(* IEC 61131-3 sources: TIA2AX/tests/test_projects/expected/HW_2000482_V18/6A1_AS17, 6 files *)

(* ---- HwInputs.st ---- *)
TYPE
	HwInputs : STRUCT
		_6A2_AS17_6A3 AT %B0 : WORD;
		_6A2_AS17_6A4 AT %B2 : WORD;
		_6A2_AS17_6A13 AT %B113 : ARRAY[0..31] OF BYTE;
		_6A2_AS17_6A20 AT %B30 : ARRAY[0..7] OF BYTE;
		HousingReader_AS17_Handshake_and_General_Error_Status_Bits_1 AT %B51 : BYTE;
		HousingReader_AS17_BUSY_Status_Bits_1 AT %B52 : BYTE;
		HousingReader_AS17_Completion_Status_Bits_1 AT %B53 : BYTE;
		HousingReader_AS17_Error_Status_Bits_1 AT %B54 : BYTE;
		HousingReader_AS17_Terminal_Status_Bits_1 AT %B55 : BYTE;
		HousingReader_AS17_Unstable_Read_Status_Bits_1 AT %B56 : BYTE;
		HousingReader_AS17_Matching_Level_and_Total_Evaluation_Grade_Status_1 AT %B57 : ARRAY[0..7] OF BYTE;
		HousingReader_AS17_Operation_Result_Status_1 AT %B87 : ARRAY[0..19] OF BYTE;
		HousingReader_AS17_Read_Data_128Byte_1 AT %B229 : ARRAY[0..135] OF BYTE;
		SEW_AS_1_Drive_1x3PD_1 AT %B107 : ARRAY[0..5] OF BYTE;
		Glue_DI_16_bytes_1 AT %B65 : ARRAY[0..15] OF BYTE;
		wp12_wp12 AT %B4 : BYTE;
	END_STRUCT;
END_TYPE

(* ---- HwOutputs.st ---- *)
TYPE
	HwOutputs : STRUCT
		_6A2_AS17_6A5 AT %B0 : WORD;
		_6A2_AS17_6A6 AT %B2 : WORD;
		_6A2_AS17_6A13 AT %B87 : ARRAY[0..31] OF BYTE;
		HousingReader_AS17_Latch_and_Error_Clear_Control_Bits_1 AT %B6 : BYTE;
		HousingReader_AS17_Operation_instruction_Control_Bits_1 AT %B7 : BYTE;
		HousingReader_AS17_Completion_Clear_Control_Bits_1 AT %B12 : BYTE;
		HousingReader_AS17_Parameter_Bank_Number_1 AT %B51 : WORD;
		HousingReader_AS17_User_Data_128Byte_1 AT %B193 : ARRAY[0..129] OF BYTE;
		CPX_PneuOst_AS17_MPA1S_VMPA1_FB_EMS_8_8DO_1 AT %B13 : BYTE;
		CPX_PneuOst_AS17_MPA1S_VMPA1_FB_EMS_8_8DO_2 AT %B183 : BYTE;
		CPX_PneuOst_AS17_MPA1S_VMPA1_FB_EMS_8_8DO_3 AT %B184 : BYTE;
		CPX_PneuOst_AS17_MPA1S_VMPA1_FB_EMS_8_8DO_4 AT %B185 : BYTE;
		CPX_PneuOst_AS17_MPA1G_VMPA1_FB_EMG_8_8DO_1 AT %B4 : BYTE;
		SEW_AS_1_Drive_1x3PD_1 AT %B69 : ARRAY[0..5] OF BYTE;
		Glue_DO_16_bytes_1 AT %B30 : ARRAY[0..15] OF BYTE;
	END_STRUCT;
END_TYPE

(* ---- PlcInputs.st ---- *)
TYPE
	PlcInputs : STRUCT
		_6A2_AS17_6A3 : WORD;
		_6A2_AS17_6A4 : WORD;
		_6A2_AS17_6A13 : ARRAY[0..31] OF BYTE;
		_6A2_AS17_6A20 : ARRAY[0..7] OF BYTE;
		HousingReader_AS17_Handshake_and_General_Error_Status_Bits_1 : BYTE;
		HousingReader_AS17_BUSY_Status_Bits_1 : BYTE;
		HousingReader_AS17_Completion_Status_Bits_1 : BYTE;
		HousingReader_AS17_Error_Status_Bits_1 : BYTE;
		HousingReader_AS17_Terminal_Status_Bits_1 : BYTE;
		HousingReader_AS17_Unstable_Read_Status_Bits_1 : BYTE;
		HousingReader_AS17_Matching_Level_and_Total_Evaluation_Grade_Status_1 : ARRAY[0..7] OF BYTE;
		HousingReader_AS17_Operation_Result_Status_1 : ARRAY[0..19] OF BYTE;
		HousingReader_AS17_Read_Data_128Byte_1 : ARRAY[0..135] OF BYTE;
		SEW_AS_1_Drive_1x3PD_1 : ARRAY[0..5] OF BYTE;
		Glue_DI_16_bytes_1 : ARRAY[0..15] OF BYTE;
		wp12_wp12 : BYTE;
	END_STRUCT;
END_TYPE

(* ---- PlcOutputs.st ---- *)
TYPE
	PlcOutputs : STRUCT
		_6A2_AS17_6A5 : WORD;
		_6A2_AS17_6A6 : WORD;
		_6A2_AS17_6A13 : ARRAY[0..31] OF BYTE;
		HousingReader_AS17_Latch_and_Error_Clear_Control_Bits_1 : BYTE;
		HousingReader_AS17_Operation_instruction_Control_Bits_1 : BYTE;
		HousingReader_AS17_Completion_Clear_Control_Bits_1 : BYTE;
		HousingReader_AS17_Parameter_Bank_Number_1 : WORD;
		HousingReader_AS17_User_Data_128Byte_1 : ARRAY[0..129] OF BYTE;
		CPX_PneuOst_AS17_MPA1S_VMPA1_FB_EMS_8_8DO_1 : BYTE;
		CPX_PneuOst_AS17_MPA1S_VMPA1_FB_EMS_8_8DO_2 : BYTE;
		CPX_PneuOst_AS17_MPA1S_VMPA1_FB_EMS_8_8DO_3 : BYTE;
		CPX_PneuOst_AS17_MPA1S_VMPA1_FB_EMS_8_8DO_4 : BYTE;
		CPX_PneuOst_AS17_MPA1G_VMPA1_FB_EMG_8_8DO_1 : BYTE;
		SEW_AS_1_Drive_1x3PD_1 : ARRAY[0..5] OF BYTE;
		Glue_DO_16_bytes_1 : ARRAY[0..15] OF BYTE;
	END_STRUCT;
END_TYPE

(* ---- CopyInputs.st ---- *)
FUNCTION CopyInputs
	VAR_EXTERNAL
		HwInputs : HwInputs;
		PlcInputs : PlcInputs;
	END_VAR
	PlcInputs._6A2_AS17_6A3 := HwInputs._6A2_AS17_6A3;
	PlcInputs._6A2_AS17_6A4 := HwInputs._6A2_AS17_6A4;
	PlcInputs._6A2_AS17_6A13[0] := HwInputs._6A2_AS17_6A13[0];
	PlcInputs._6A2_AS17_6A13[1] := HwInputs._6A2_AS17_6A13[1];
	PlcInputs._6A2_AS17_6A13[2] := HwInputs._6A2_AS17_6A13[2];
	PlcInputs._6A2_AS17_6A13[3] := HwInputs._6A2_AS17_6A13[3];
	PlcInputs._6A2_AS17_6A13[4] := HwInputs._6A2_AS17_6A13[4];
	PlcInputs._6A2_AS17_6A13[5] := HwInputs._6A2_AS17_6A13[5];
	PlcInputs._6A2_AS17_6A13[6] := HwInputs._6A2_AS17_6A13[6];
	PlcInputs._6A2_AS17_6A13[7] := HwInputs._6A2_AS17_6A13[7];
	PlcInputs._6A2_AS17_6A13[8] := HwInputs._6A2_AS17_6A13[8];
	PlcInputs._6A2_AS17_6A13[9] := HwInputs._6A2_AS17_6A13[9];
	PlcInputs._6A2_AS17_6A13[10] := HwInputs._6A2_AS17_6A13[10];
	PlcInputs._6A2_AS17_6A13[11] := HwInputs._6A2_AS17_6A13[11];
	PlcInputs._6A2_AS17_6A13[12] := HwInputs._6A2_AS17_6A13[12];
	PlcInputs._6A2_AS17_6A13[13] := HwInputs._6A2_AS17_6A13[13];
	PlcInputs._6A2_AS17_6A13[14] := HwInputs._6A2_AS17_6A13[14];
	PlcInputs._6A2_AS17_6A13[15] := HwInputs._6A2_AS17_6A13[15];
	PlcInputs._6A2_AS17_6A13[16] := HwInputs._6A2_AS17_6A13[16];
	PlcInputs._6A2_AS17_6A13[17] := HwInputs._6A2_AS17_6A13[17];
	PlcInputs._6A2_AS17_6A13[18] := HwInputs._6A2_AS17_6A13[18];
	PlcInputs._6A2_AS17_6A13[19] := HwInputs._6A2_AS17_6A13[19];
	PlcInputs._6A2_AS17_6A13[20] := HwInputs._6A2_AS17_6A13[20];
	PlcInputs._6A2_AS17_6A13[21] := HwInputs._6A2_AS17_6A13[21];
	PlcInputs._6A2_AS17_6A13[22] := HwInputs._6A2_AS17_6A13[22];
	PlcInputs._6A2_AS17_6A13[23] := HwInputs._6A2_AS17_6A13[23];
	PlcInputs._6A2_AS17_6A13[24] := HwInputs._6A2_AS17_6A13[24];
	PlcInputs._6A2_AS17_6A13[25] := HwInputs._6A2_AS17_6A13[25];
	PlcInputs._6A2_AS17_6A13[26] := HwInputs._6A2_AS17_6A13[26];
	PlcInputs._6A2_AS17_6A13[27] := HwInputs._6A2_AS17_6A13[27];
	PlcInputs._6A2_AS17_6A13[28] := HwInputs._6A2_AS17_6A13[28];
	PlcInputs._6A2_AS17_6A13[29] := HwInputs._6A2_AS17_6A13[29];
	PlcInputs._6A2_AS17_6A13[30] := HwInputs._6A2_AS17_6A13[30];
	PlcInputs._6A2_AS17_6A13[31] := HwInputs._6A2_AS17_6A13[31];
	PlcInputs._6A2_AS17_6A20[0] := HwInputs._6A2_AS17_6A20[0];
	PlcInputs._6A2_AS17_6A20[1] := HwInputs._6A2_AS17_6A20[1];
	PlcInputs._6A2_AS17_6A20[2] := HwInputs._6A2_AS17_6A20[2];
	PlcInputs._6A2_AS17_6A20[3] := HwInputs._6A2_AS17_6A20[3];
	PlcInputs._6A2_AS17_6A20[4] := HwInputs._6A2_AS17_6A20[4];
	PlcInputs._6A2_AS17_6A20[5] := HwInputs._6A2_AS17_6A20[5];
	PlcInputs._6A2_AS17_6A20[6] := HwInputs._6A2_AS17_6A20[6];
	PlcInputs._6A2_AS17_6A20[7] := HwInputs._6A2_AS17_6A20[7];
	PlcInputs.HousingReader_AS17_Handshake_and_General_Error_Status_Bits_1 := HwInputs.HousingReader_AS17_Handshake_and_General_Error_Status_Bits_1;
	PlcInputs.HousingReader_AS17_BUSY_Status_Bits_1 := HwInputs.HousingReader_AS17_BUSY_Status_Bits_1;
	PlcInputs.HousingReader_AS17_Completion_Status_Bits_1 := HwInputs.HousingReader_AS17_Completion_Status_Bits_1;
	PlcInputs.HousingReader_AS17_Error_Status_Bits_1 := HwInputs.HousingReader_AS17_Error_Status_Bits_1;
	PlcInputs.HousingReader_AS17_Terminal_Status_Bits_1 := HwInputs.HousingReader_AS17_Terminal_Status_Bits_1;
	PlcInputs.HousingReader_AS17_Unstable_Read_Status_Bits_1 := HwInputs.HousingReader_AS17_Unstable_Read_Status_Bits_1;
	PlcInputs.HousingReader_AS17_Matching_Level_and_Total_Evaluation_Grade_Status_1[0] := HwInputs.HousingReader_AS17_Matching_Level_and_Total_Evaluation_Grade_Status_1[0];
	PlcInputs.HousingReader_AS17_Matching_Level_and_Total_Evaluation_Grade_Status_1[1] := HwInputs.HousingReader_AS17_Matching_Level_and_Total_Evaluation_Grade_Status_1[1];
	PlcInputs.HousingReader_AS17_Matching_Level_and_Total_Evaluation_Grade_Status_1[2] := HwInputs.HousingReader_AS17_Matching_Level_and_Total_Evaluation_Grade_Status_1[2];
	PlcInputs.HousingReader_AS17_Matching_Level_and_Total_Evaluation_Grade_Status_1[3] := HwInputs.HousingReader_AS17_Matching_Level_and_Total_Evaluation_Grade_Status_1[3];
	PlcInputs.HousingReader_AS17_Matching_Level_and_Total_Evaluation_Grade_Status_1[4] := HwInputs.HousingReader_AS17_Matching_Level_and_Total_Evaluation_Grade_Status_1[4];
	PlcInputs.HousingReader_AS17_Matching_Level_and_Total_Evaluation_Grade_Status_1[5] := HwInputs.HousingReader_AS17_Matching_Level_and_Total_Evaluation_Grade_Status_1[5];
	PlcInputs.HousingReader_AS17_Matching_Level_and_Total_Evaluation_Grade_Status_1[6] := HwInputs.HousingReader_AS17_Matching_Level_and_Total_Evaluation_Grade_Status_1[6];
	PlcInputs.HousingReader_AS17_Matching_Level_and_Total_Evaluation_Grade_Status_1[7] := HwInputs.HousingReader_AS17_Matching_Level_and_Total_Evaluation_Grade_Status_1[7];
	PlcInputs.HousingReader_AS17_Operation_Result_Status_1[0] := HwInputs.HousingReader_AS17_Operation_Result_Status_1[0];
	PlcInputs.HousingReader_AS17_Operation_Result_Status_1[1] := HwInputs.HousingReader_AS17_Operation_Result_Status_1[1];
	PlcInputs.HousingReader_AS17_Operation_Result_Status_1[2] := HwInputs.HousingReader_AS17_Operation_Result_Status_1[2];
	PlcInputs.HousingReader_AS17_Operation_Result_Status_1[3] := HwInputs.HousingReader_AS17_Operation_Result_Status_1[3];
	PlcInputs.HousingReader_AS17_Operation_Result_Status_1[4] := HwInputs.HousingReader_AS17_Operation_Result_Status_1[4];
	PlcInputs.HousingReader_AS17_Operation_Result_Status_1[5] := HwInputs.HousingReader_AS17_Operation_Result_Status_1[5];
	PlcInputs.HousingReader_AS17_Operation_Result_Status_1[6] := HwInputs.HousingReader_AS17_Operation_Result_Status_1[6];
	PlcInputs.HousingReader_AS17_Operation_Result_Status_1[7] := HwInputs.HousingReader_AS17_Operation_Result_Status_1[7];
	PlcInputs.HousingReader_AS17_Operation_Result_Status_1[8] := HwInputs.HousingReader_AS17_Operation_Result_Status_1[8];
	PlcInputs.HousingReader_AS17_Operation_Result_Status_1[9] := HwInputs.HousingReader_AS17_Operation_Result_Status_1[9];
	PlcInputs.HousingReader_AS17_Operation_Result_Status_1[10] := HwInputs.HousingReader_AS17_Operation_Result_Status_1[10];
	PlcInputs.HousingReader_AS17_Operation_Result_Status_1[11] := HwInputs.HousingReader_AS17_Operation_Result_Status_1[11];
	PlcInputs.HousingReader_AS17_Operation_Result_Status_1[12] := HwInputs.HousingReader_AS17_Operation_Result_Status_1[12];
	PlcInputs.HousingReader_AS17_Operation_Result_Status_1[13] := HwInputs.HousingReader_AS17_Operation_Result_Status_1[13];
	PlcInputs.HousingReader_AS17_Operation_Result_Status_1[14] := HwInputs.HousingReader_AS17_Operation_Result_Status_1[14];
	PlcInputs.HousingReader_AS17_Operation_Result_Status_1[15] := HwInputs.HousingReader_AS17_Operation_Result_Status_1[15];
	PlcInputs.HousingReader_AS17_Operation_Result_Status_1[16] := HwInputs.HousingReader_AS17_Operation_Result_Status_1[16];
	PlcInputs.HousingReader_AS17_Operation_Result_Status_1[17] := HwInputs.HousingReader_AS17_Operation_Result_Status_1[17];
	PlcInputs.HousingReader_AS17_Operation_Result_Status_1[18] := HwInputs.HousingReader_AS17_Operation_Result_Status_1[18];
	PlcInputs.HousingReader_AS17_Operation_Result_Status_1[19] := HwInputs.HousingReader_AS17_Operation_Result_Status_1[19];
	PlcInputs.HousingReader_AS17_Read_Data_128Byte_1[0] := HwInputs.HousingReader_AS17_Read_Data_128Byte_1[0];
	PlcInputs.HousingReader_AS17_Read_Data_128Byte_1[1] := HwInputs.HousingReader_AS17_Read_Data_128Byte_1[1];
	PlcInputs.HousingReader_AS17_Read_Data_128Byte_1[2] := HwInputs.HousingReader_AS17_Read_Data_128Byte_1[2];
	PlcInputs.HousingReader_AS17_Read_Data_128Byte_1[3] := HwInputs.HousingReader_AS17_Read_Data_128Byte_1[3];
	PlcInputs.HousingReader_AS17_Read_Data_128Byte_1[4] := HwInputs.HousingReader_AS17_Read_Data_128Byte_1[4];
	PlcInputs.HousingReader_AS17_Read_Data_128Byte_1[5] := HwInputs.HousingReader_AS17_Read_Data_128Byte_1[5];
	PlcInputs.HousingReader_AS17_Read_Data_128Byte_1[6] := HwInputs.HousingReader_AS17_Read_Data_128Byte_1[6];
	PlcInputs.HousingReader_AS17_Read_Data_128Byte_1[7] := HwInputs.HousingReader_AS17_Read_Data_128Byte_1[7];
	PlcInputs.HousingReader_AS17_Read_Data_128Byte_1[8] := HwInputs.HousingReader_AS17_Read_Data_128Byte_1[8];
	PlcInputs.HousingReader_AS17_Read_Data_128Byte_1[9] := HwInputs.HousingReader_AS17_Read_Data_128Byte_1[9];
	PlcInputs.HousingReader_AS17_Read_Data_128Byte_1[10] := HwInputs.HousingReader_AS17_Read_Data_128Byte_1[10];
	PlcInputs.HousingReader_AS17_Read_Data_128Byte_1[11] := HwInputs.HousingReader_AS17_Read_Data_128Byte_1[11];
	PlcInputs.HousingReader_AS17_Read_Data_128Byte_1[12] := HwInputs.HousingReader_AS17_Read_Data_128Byte_1[12];
	PlcInputs.HousingReader_AS17_Read_Data_128Byte_1[13] := HwInputs.HousingReader_AS17_Read_Data_128Byte_1[13];
	PlcInputs.HousingReader_AS17_Read_Data_128Byte_1[14] := HwInputs.HousingReader_AS17_Read_Data_128Byte_1[14];
	PlcInputs.HousingReader_AS17_Read_Data_128Byte_1[15] := HwInputs.HousingReader_AS17_Read_Data_128Byte_1[15];
	PlcInputs.HousingReader_AS17_Read_Data_128Byte_1[16] := HwInputs.HousingReader_AS17_Read_Data_128Byte_1[16];
	PlcInputs.HousingReader_AS17_Read_Data_128Byte_1[17] := HwInputs.HousingReader_AS17_Read_Data_128Byte_1[17];
	PlcInputs.HousingReader_AS17_Read_Data_128Byte_1[18] := HwInputs.HousingReader_AS17_Read_Data_128Byte_1[18];
	PlcInputs.HousingReader_AS17_Read_Data_128Byte_1[19] := HwInputs.HousingReader_AS17_Read_Data_128Byte_1[19];
	PlcInputs.HousingReader_AS17_Read_Data_128Byte_1[20] := HwInputs.HousingReader_AS17_Read_Data_128Byte_1[20];
	PlcInputs.HousingReader_AS17_Read_Data_128Byte_1[21] := HwInputs.HousingReader_AS17_Read_Data_128Byte_1[21];
	PlcInputs.HousingReader_AS17_Read_Data_128Byte_1[22] := HwInputs.HousingReader_AS17_Read_Data_128Byte_1[22];
	PlcInputs.HousingReader_AS17_Read_Data_128Byte_1[23] := HwInputs.HousingReader_AS17_Read_Data_128Byte_1[23];
	PlcInputs.HousingReader_AS17_Read_Data_128Byte_1[24] := HwInputs.HousingReader_AS17_Read_Data_128Byte_1[24];
	PlcInputs.HousingReader_AS17_Read_Data_128Byte_1[25] := HwInputs.HousingReader_AS17_Read_Data_128Byte_1[25];
	PlcInputs.HousingReader_AS17_Read_Data_128Byte_1[26] := HwInputs.HousingReader_AS17_Read_Data_128Byte_1[26];
	PlcInputs.HousingReader_AS17_Read_Data_128Byte_1[27] := HwInputs.HousingReader_AS17_Read_Data_128Byte_1[27];
	PlcInputs.HousingReader_AS17_Read_Data_128Byte_1[28] := HwInputs.HousingReader_AS17_Read_Data_128Byte_1[28];
	PlcInputs.HousingReader_AS17_Read_Data_128Byte_1[29] := HwInputs.HousingReader_AS17_Read_Data_128Byte_1[29];
	PlcInputs.HousingReader_AS17_Read_Data_128Byte_1[30] := HwInputs.HousingReader_AS17_Read_Data_128Byte_1[30];
	PlcInputs.HousingReader_AS17_Read_Data_128Byte_1[31] := HwInputs.HousingReader_AS17_Read_Data_128Byte_1[31];
	PlcInputs.HousingReader_AS17_Read_Data_128Byte_1[32] := HwInputs.HousingReader_AS17_Read_Data_128Byte_1[32];
	PlcInputs.HousingReader_AS17_Read_Data_128Byte_1[33] := HwInputs.HousingReader_AS17_Read_Data_128Byte_1[33];
	PlcInputs.HousingReader_AS17_Read_Data_128Byte_1[34] := HwInputs.HousingReader_AS17_Read_Data_128Byte_1[34];
	PlcInputs.HousingReader_AS17_Read_Data_128Byte_1[35] := HwInputs.HousingReader_AS17_Read_Data_128Byte_1[35];
	PlcInputs.HousingReader_AS17_Read_Data_128Byte_1[36] := HwInputs.HousingReader_AS17_Read_Data_128Byte_1[36];
	PlcInputs.HousingReader_AS17_Read_Data_128Byte_1[37] := HwInputs.HousingReader_AS17_Read_Data_128Byte_1[37];
	PlcInputs.HousingReader_AS17_Read_Data_128Byte_1[38] := HwInputs.HousingReader_AS17_Read_Data_128Byte_1[38];
	PlcInputs.HousingReader_AS17_Read_Data_128Byte_1[39] := HwInputs.HousingReader_AS17_Read_Data_128Byte_1[39];
	PlcInputs.HousingReader_AS17_Read_Data_128Byte_1[40] := HwInputs.HousingReader_AS17_Read_Data_128Byte_1[40];
	PlcInputs.HousingReader_AS17_Read_Data_128Byte_1[41] := HwInputs.HousingReader_AS17_Read_Data_128Byte_1[41];
	PlcInputs.HousingReader_AS17_Read_Data_128Byte_1[42] := HwInputs.HousingReader_AS17_Read_Data_128Byte_1[42];
	PlcInputs.HousingReader_AS17_Read_Data_128Byte_1[43] := HwInputs.HousingReader_AS17_Read_Data_128Byte_1[43];
	PlcInputs.HousingReader_AS17_Read_Data_128Byte_1[44] := HwInputs.HousingReader_AS17_Read_Data_128Byte_1[44];
	PlcInputs.HousingReader_AS17_Read_Data_128Byte_1[45] := HwInputs.HousingReader_AS17_Read_Data_128Byte_1[45];
	PlcInputs.HousingReader_AS17_Read_Data_128Byte_1[46] := HwInputs.HousingReader_AS17_Read_Data_128Byte_1[46];
	PlcInputs.HousingReader_AS17_Read_Data_128Byte_1[47] := HwInputs.HousingReader_AS17_Read_Data_128Byte_1[47];
	PlcInputs.HousingReader_AS17_Read_Data_128Byte_1[48] := HwInputs.HousingReader_AS17_Read_Data_128Byte_1[48];
	PlcInputs.HousingReader_AS17_Read_Data_128Byte_1[49] := HwInputs.HousingReader_AS17_Read_Data_128Byte_1[49];
	PlcInputs.HousingReader_AS17_Read_Data_128Byte_1[50] := HwInputs.HousingReader_AS17_Read_Data_128Byte_1[50];
	PlcInputs.HousingReader_AS17_Read_Data_128Byte_1[51] := HwInputs.HousingReader_AS17_Read_Data_128Byte_1[51];
	PlcInputs.HousingReader_AS17_Read_Data_128Byte_1[52] := HwInputs.HousingReader_AS17_Read_Data_128Byte_1[52];
	PlcInputs.HousingReader_AS17_Read_Data_128Byte_1[53] := HwInputs.HousingReader_AS17_Read_Data_128Byte_1[53];
	PlcInputs.HousingReader_AS17_Read_Data_128Byte_1[54] := HwInputs.HousingReader_AS17_Read_Data_128Byte_1[54];
	PlcInputs.HousingReader_AS17_Read_Data_128Byte_1[55] := HwInputs.HousingReader_AS17_Read_Data_128Byte_1[55];
	PlcInputs.HousingReader_AS17_Read_Data_128Byte_1[56] := HwInputs.HousingReader_AS17_Read_Data_128Byte_1[56];
	PlcInputs.HousingReader_AS17_Read_Data_128Byte_1[57] := HwInputs.HousingReader_AS17_Read_Data_128Byte_1[57];
	PlcInputs.HousingReader_AS17_Read_Data_128Byte_1[58] := HwInputs.HousingReader_AS17_Read_Data_128Byte_1[58];
	PlcInputs.HousingReader_AS17_Read_Data_128Byte_1[59] := HwInputs.HousingReader_AS17_Read_Data_128Byte_1[59];
	PlcInputs.HousingReader_AS17_Read_Data_128Byte_1[60] := HwInputs.HousingReader_AS17_Read_Data_128Byte_1[60];
	PlcInputs.HousingReader_AS17_Read_Data_128Byte_1[61] := HwInputs.HousingReader_AS17_Read_Data_128Byte_1[61];
	PlcInputs.HousingReader_AS17_Read_Data_128Byte_1[62] := HwInputs.HousingReader_AS17_Read_Data_128Byte_1[62];
	PlcInputs.HousingReader_AS17_Read_Data_128Byte_1[63] := HwInputs.HousingReader_AS17_Read_Data_128Byte_1[63];
	PlcInputs.HousingReader_AS17_Read_Data_128Byte_1[64] := HwInputs.HousingReader_AS17_Read_Data_128Byte_1[64];
	PlcInputs.HousingReader_AS17_Read_Data_128Byte_1[65] := HwInputs.HousingReader_AS17_Read_Data_128Byte_1[65];
	PlcInputs.HousingReader_AS17_Read_Data_128Byte_1[66] := HwInputs.HousingReader_AS17_Read_Data_128Byte_1[66];
	PlcInputs.HousingReader_AS17_Read_Data_128Byte_1[67] := HwInputs.HousingReader_AS17_Read_Data_128Byte_1[67];
	PlcInputs.HousingReader_AS17_Read_Data_128Byte_1[68] := HwInputs.HousingReader_AS17_Read_Data_128Byte_1[68];
	PlcInputs.HousingReader_AS17_Read_Data_128Byte_1[69] := HwInputs.HousingReader_AS17_Read_Data_128Byte_1[69];
	PlcInputs.HousingReader_AS17_Read_Data_128Byte_1[70] := HwInputs.HousingReader_AS17_Read_Data_128Byte_1[70];
	PlcInputs.HousingReader_AS17_Read_Data_128Byte_1[71] := HwInputs.HousingReader_AS17_Read_Data_128Byte_1[71];
	PlcInputs.HousingReader_AS17_Read_Data_128Byte_1[72] := HwInputs.HousingReader_AS17_Read_Data_128Byte_1[72];
	PlcInputs.HousingReader_AS17_Read_Data_128Byte_1[73] := HwInputs.HousingReader_AS17_Read_Data_128Byte_1[73];
	PlcInputs.HousingReader_AS17_Read_Data_128Byte_1[74] := HwInputs.HousingReader_AS17_Read_Data_128Byte_1[74];
	PlcInputs.HousingReader_AS17_Read_Data_128Byte_1[75] := HwInputs.HousingReader_AS17_Read_Data_128Byte_1[75];
	PlcInputs.HousingReader_AS17_Read_Data_128Byte_1[76] := HwInputs.HousingReader_AS17_Read_Data_128Byte_1[76];
	PlcInputs.HousingReader_AS17_Read_Data_128Byte_1[77] := HwInputs.HousingReader_AS17_Read_Data_128Byte_1[77];
	PlcInputs.HousingReader_AS17_Read_Data_128Byte_1[78] := HwInputs.HousingReader_AS17_Read_Data_128Byte_1[78];
	PlcInputs.HousingReader_AS17_Read_Data_128Byte_1[79] := HwInputs.HousingReader_AS17_Read_Data_128Byte_1[79];
	PlcInputs.HousingReader_AS17_Read_Data_128Byte_1[80] := HwInputs.HousingReader_AS17_Read_Data_128Byte_1[80];
	PlcInputs.HousingReader_AS17_Read_Data_128Byte_1[81] := HwInputs.HousingReader_AS17_Read_Data_128Byte_1[81];
	PlcInputs.HousingReader_AS17_Read_Data_128Byte_1[82] := HwInputs.HousingReader_AS17_Read_Data_128Byte_1[82];
	PlcInputs.HousingReader_AS17_Read_Data_128Byte_1[83] := HwInputs.HousingReader_AS17_Read_Data_128Byte_1[83];
	PlcInputs.HousingReader_AS17_Read_Data_128Byte_1[84] := HwInputs.HousingReader_AS17_Read_Data_128Byte_1[84];
	PlcInputs.HousingReader_AS17_Read_Data_128Byte_1[85] := HwInputs.HousingReader_AS17_Read_Data_128Byte_1[85];
	PlcInputs.HousingReader_AS17_Read_Data_128Byte_1[86] := HwInputs.HousingReader_AS17_Read_Data_128Byte_1[86];
	PlcInputs.HousingReader_AS17_Read_Data_128Byte_1[87] := HwInputs.HousingReader_AS17_Read_Data_128Byte_1[87];
	PlcInputs.HousingReader_AS17_Read_Data_128Byte_1[88] := HwInputs.HousingReader_AS17_Read_Data_128Byte_1[88];
	PlcInputs.HousingReader_AS17_Read_Data_128Byte_1[89] := HwInputs.HousingReader_AS17_Read_Data_128Byte_1[89];
	PlcInputs.HousingReader_AS17_Read_Data_128Byte_1[90] := HwInputs.HousingReader_AS17_Read_Data_128Byte_1[90];
	PlcInputs.HousingReader_AS17_Read_Data_128Byte_1[91] := HwInputs.HousingReader_AS17_Read_Data_128Byte_1[91];
	PlcInputs.HousingReader_AS17_Read_Data_128Byte_1[92] := HwInputs.HousingReader_AS17_Read_Data_128Byte_1[92];
	PlcInputs.HousingReader_AS17_Read_Data_128Byte_1[93] := HwInputs.HousingReader_AS17_Read_Data_128Byte_1[93];
	PlcInputs.HousingReader_AS17_Read_Data_128Byte_1[94] := HwInputs.HousingReader_AS17_Read_Data_128Byte_1[94];
	PlcInputs.HousingReader_AS17_Read_Data_128Byte_1[95] := HwInputs.HousingReader_AS17_Read_Data_128Byte_1[95];
	PlcInputs.HousingReader_AS17_Read_Data_128Byte_1[96] := HwInputs.HousingReader_AS17_Read_Data_128Byte_1[96];
	PlcInputs.HousingReader_AS17_Read_Data_128Byte_1[97] := HwInputs.HousingReader_AS17_Read_Data_128Byte_1[97];
	PlcInputs.HousingReader_AS17_Read_Data_128Byte_1[98] := HwInputs.HousingReader_AS17_Read_Data_128Byte_1[98];
	PlcInputs.HousingReader_AS17_Read_Data_128Byte_1[99] := HwInputs.HousingReader_AS17_Read_Data_128Byte_1[99];
	PlcInputs.HousingReader_AS17_Read_Data_128Byte_1[100] := HwInputs.HousingReader_AS17_Read_Data_128Byte_1[100];
	PlcInputs.HousingReader_AS17_Read_Data_128Byte_1[101] := HwInputs.HousingReader_AS17_Read_Data_128Byte_1[101];
	PlcInputs.HousingReader_AS17_Read_Data_128Byte_1[102] := HwInputs.HousingReader_AS17_Read_Data_128Byte_1[102];
	PlcInputs.HousingReader_AS17_Read_Data_128Byte_1[103] := HwInputs.HousingReader_AS17_Read_Data_128Byte_1[103];
	PlcInputs.HousingReader_AS17_Read_Data_128Byte_1[104] := HwInputs.HousingReader_AS17_Read_Data_128Byte_1[104];
	PlcInputs.HousingReader_AS17_Read_Data_128Byte_1[105] := HwInputs.HousingReader_AS17_Read_Data_128Byte_1[105];
	PlcInputs.HousingReader_AS17_Read_Data_128Byte_1[106] := HwInputs.HousingReader_AS17_Read_Data_128Byte_1[106];
	PlcInputs.HousingReader_AS17_Read_Data_128Byte_1[107] := HwInputs.HousingReader_AS17_Read_Data_128Byte_1[107];
	PlcInputs.HousingReader_AS17_Read_Data_128Byte_1[108] := HwInputs.HousingReader_AS17_Read_Data_128Byte_1[108];
	PlcInputs.HousingReader_AS17_Read_Data_128Byte_1[109] := HwInputs.HousingReader_AS17_Read_Data_128Byte_1[109];
	PlcInputs.HousingReader_AS17_Read_Data_128Byte_1[110] := HwInputs.HousingReader_AS17_Read_Data_128Byte_1[110];
	PlcInputs.HousingReader_AS17_Read_Data_128Byte_1[111] := HwInputs.HousingReader_AS17_Read_Data_128Byte_1[111];
	PlcInputs.HousingReader_AS17_Read_Data_128Byte_1[112] := HwInputs.HousingReader_AS17_Read_Data_128Byte_1[112];
	PlcInputs.HousingReader_AS17_Read_Data_128Byte_1[113] := HwInputs.HousingReader_AS17_Read_Data_128Byte_1[113];
	PlcInputs.HousingReader_AS17_Read_Data_128Byte_1[114] := HwInputs.HousingReader_AS17_Read_Data_128Byte_1[114];
	PlcInputs.HousingReader_AS17_Read_Data_128Byte_1[115] := HwInputs.HousingReader_AS17_Read_Data_128Byte_1[115];
	PlcInputs.HousingReader_AS17_Read_Data_128Byte_1[116] := HwInputs.HousingReader_AS17_Read_Data_128Byte_1[116];
	PlcInputs.HousingReader_AS17_Read_Data_128Byte_1[117] := HwInputs.HousingReader_AS17_Read_Data_128Byte_1[117];
	PlcInputs.HousingReader_AS17_Read_Data_128Byte_1[118] := HwInputs.HousingReader_AS17_Read_Data_128Byte_1[118];
	PlcInputs.HousingReader_AS17_Read_Data_128Byte_1[119] := HwInputs.HousingReader_AS17_Read_Data_128Byte_1[119];
	PlcInputs.HousingReader_AS17_Read_Data_128Byte_1[120] := HwInputs.HousingReader_AS17_Read_Data_128Byte_1[120];
	PlcInputs.HousingReader_AS17_Read_Data_128Byte_1[121] := HwInputs.HousingReader_AS17_Read_Data_128Byte_1[121];
	PlcInputs.HousingReader_AS17_Read_Data_128Byte_1[122] := HwInputs.HousingReader_AS17_Read_Data_128Byte_1[122];
	PlcInputs.HousingReader_AS17_Read_Data_128Byte_1[123] := HwInputs.HousingReader_AS17_Read_Data_128Byte_1[123];
	PlcInputs.HousingReader_AS17_Read_Data_128Byte_1[124] := HwInputs.HousingReader_AS17_Read_Data_128Byte_1[124];
	PlcInputs.HousingReader_AS17_Read_Data_128Byte_1[125] := HwInputs.HousingReader_AS17_Read_Data_128Byte_1[125];
	PlcInputs.HousingReader_AS17_Read_Data_128Byte_1[126] := HwInputs.HousingReader_AS17_Read_Data_128Byte_1[126];
	PlcInputs.HousingReader_AS17_Read_Data_128Byte_1[127] := HwInputs.HousingReader_AS17_Read_Data_128Byte_1[127];
	PlcInputs.HousingReader_AS17_Read_Data_128Byte_1[128] := HwInputs.HousingReader_AS17_Read_Data_128Byte_1[128];
	PlcInputs.HousingReader_AS17_Read_Data_128Byte_1[129] := HwInputs.HousingReader_AS17_Read_Data_128Byte_1[129];
	PlcInputs.HousingReader_AS17_Read_Data_128Byte_1[130] := HwInputs.HousingReader_AS17_Read_Data_128Byte_1[130];
	PlcInputs.HousingReader_AS17_Read_Data_128Byte_1[131] := HwInputs.HousingReader_AS17_Read_Data_128Byte_1[131];
	PlcInputs.HousingReader_AS17_Read_Data_128Byte_1[132] := HwInputs.HousingReader_AS17_Read_Data_128Byte_1[132];
	PlcInputs.HousingReader_AS17_Read_Data_128Byte_1[133] := HwInputs.HousingReader_AS17_Read_Data_128Byte_1[133];
	PlcInputs.HousingReader_AS17_Read_Data_128Byte_1[134] := HwInputs.HousingReader_AS17_Read_Data_128Byte_1[134];
	PlcInputs.HousingReader_AS17_Read_Data_128Byte_1[135] := HwInputs.HousingReader_AS17_Read_Data_128Byte_1[135];
	PlcInputs.SEW_AS_1_Drive_1x3PD_1[0] := HwInputs.SEW_AS_1_Drive_1x3PD_1[0];
	PlcInputs.SEW_AS_1_Drive_1x3PD_1[1] := HwInputs.SEW_AS_1_Drive_1x3PD_1[1];
	PlcInputs.SEW_AS_1_Drive_1x3PD_1[2] := HwInputs.SEW_AS_1_Drive_1x3PD_1[2];
	PlcInputs.SEW_AS_1_Drive_1x3PD_1[3] := HwInputs.SEW_AS_1_Drive_1x3PD_1[3];
	PlcInputs.SEW_AS_1_Drive_1x3PD_1[4] := HwInputs.SEW_AS_1_Drive_1x3PD_1[4];
	PlcInputs.SEW_AS_1_Drive_1x3PD_1[5] := HwInputs.SEW_AS_1_Drive_1x3PD_1[5];
	PlcInputs.Glue_DI_16_bytes_1[0] := HwInputs.Glue_DI_16_bytes_1[0];
	PlcInputs.Glue_DI_16_bytes_1[1] := HwInputs.Glue_DI_16_bytes_1[1];
	PlcInputs.Glue_DI_16_bytes_1[2] := HwInputs.Glue_DI_16_bytes_1[2];
	PlcInputs.Glue_DI_16_bytes_1[3] := HwInputs.Glue_DI_16_bytes_1[3];
	PlcInputs.Glue_DI_16_bytes_1[4] := HwInputs.Glue_DI_16_bytes_1[4];
	PlcInputs.Glue_DI_16_bytes_1[5] := HwInputs.Glue_DI_16_bytes_1[5];
	PlcInputs.Glue_DI_16_bytes_1[6] := HwInputs.Glue_DI_16_bytes_1[6];
	PlcInputs.Glue_DI_16_bytes_1[7] := HwInputs.Glue_DI_16_bytes_1[7];
	PlcInputs.Glue_DI_16_bytes_1[8] := HwInputs.Glue_DI_16_bytes_1[8];
	PlcInputs.Glue_DI_16_bytes_1[9] := HwInputs.Glue_DI_16_bytes_1[9];
	PlcInputs.Glue_DI_16_bytes_1[10] := HwInputs.Glue_DI_16_bytes_1[10];
	PlcInputs.Glue_DI_16_bytes_1[11] := HwInputs.Glue_DI_16_bytes_1[11];
	PlcInputs.Glue_DI_16_bytes_1[12] := HwInputs.Glue_DI_16_bytes_1[12];
	PlcInputs.Glue_DI_16_bytes_1[13] := HwInputs.Glue_DI_16_bytes_1[13];
	PlcInputs.Glue_DI_16_bytes_1[14] := HwInputs.Glue_DI_16_bytes_1[14];
	PlcInputs.Glue_DI_16_bytes_1[15] := HwInputs.Glue_DI_16_bytes_1[15];
	PlcInputs.wp12_wp12 := HwInputs.wp12_wp12;
END_FUNCTION

(* ---- CopyOutputs.st ---- *)
FUNCTION CopyOutputs
	VAR_EXTERNAL
		HwOutputs : HwOutputs;
		PlcOutputs : PlcOutputs;
	END_VAR
	HwOutputs._6A2_AS17_6A5 := PlcOutputs._6A2_AS17_6A5;
	HwOutputs._6A2_AS17_6A6 := PlcOutputs._6A2_AS17_6A6;
	HwOutputs._6A2_AS17_6A13[0] := PlcOutputs._6A2_AS17_6A13[0];
	HwOutputs._6A2_AS17_6A13[1] := PlcOutputs._6A2_AS17_6A13[1];
	HwOutputs._6A2_AS17_6A13[2] := PlcOutputs._6A2_AS17_6A13[2];
	HwOutputs._6A2_AS17_6A13[3] := PlcOutputs._6A2_AS17_6A13[3];
	HwOutputs._6A2_AS17_6A13[4] := PlcOutputs._6A2_AS17_6A13[4];
	HwOutputs._6A2_AS17_6A13[5] := PlcOutputs._6A2_AS17_6A13[5];
	HwOutputs._6A2_AS17_6A13[6] := PlcOutputs._6A2_AS17_6A13[6];
	HwOutputs._6A2_AS17_6A13[7] := PlcOutputs._6A2_AS17_6A13[7];
	HwOutputs._6A2_AS17_6A13[8] := PlcOutputs._6A2_AS17_6A13[8];
	HwOutputs._6A2_AS17_6A13[9] := PlcOutputs._6A2_AS17_6A13[9];
	HwOutputs._6A2_AS17_6A13[10] := PlcOutputs._6A2_AS17_6A13[10];
	HwOutputs._6A2_AS17_6A13[11] := PlcOutputs._6A2_AS17_6A13[11];
	HwOutputs._6A2_AS17_6A13[12] := PlcOutputs._6A2_AS17_6A13[12];
	HwOutputs._6A2_AS17_6A13[13] := PlcOutputs._6A2_AS17_6A13[13];
	HwOutputs._6A2_AS17_6A13[14] := PlcOutputs._6A2_AS17_6A13[14];
	HwOutputs._6A2_AS17_6A13[15] := PlcOutputs._6A2_AS17_6A13[15];
	HwOutputs._6A2_AS17_6A13[16] := PlcOutputs._6A2_AS17_6A13[16];
	HwOutputs._6A2_AS17_6A13[17] := PlcOutputs._6A2_AS17_6A13[17];
	HwOutputs._6A2_AS17_6A13[18] := PlcOutputs._6A2_AS17_6A13[18];
	HwOutputs._6A2_AS17_6A13[19] := PlcOutputs._6A2_AS17_6A13[19];
	HwOutputs._6A2_AS17_6A13[20] := PlcOutputs._6A2_AS17_6A13[20];
	HwOutputs._6A2_AS17_6A13[21] := PlcOutputs._6A2_AS17_6A13[21];
	HwOutputs._6A2_AS17_6A13[22] := PlcOutputs._6A2_AS17_6A13[22];
	HwOutputs._6A2_AS17_6A13[23] := PlcOutputs._6A2_AS17_6A13[23];
	HwOutputs._6A2_AS17_6A13[24] := PlcOutputs._6A2_AS17_6A13[24];
	HwOutputs._6A2_AS17_6A13[25] := PlcOutputs._6A2_AS17_6A13[25];
	HwOutputs._6A2_AS17_6A13[26] := PlcOutputs._6A2_AS17_6A13[26];
	HwOutputs._6A2_AS17_6A13[27] := PlcOutputs._6A2_AS17_6A13[27];
	HwOutputs._6A2_AS17_6A13[28] := PlcOutputs._6A2_AS17_6A13[28];
	HwOutputs._6A2_AS17_6A13[29] := PlcOutputs._6A2_AS17_6A13[29];
	HwOutputs._6A2_AS17_6A13[30] := PlcOutputs._6A2_AS17_6A13[30];
	HwOutputs._6A2_AS17_6A13[31] := PlcOutputs._6A2_AS17_6A13[31];
	HwOutputs.HousingReader_AS17_Latch_and_Error_Clear_Control_Bits_1 := PlcOutputs.HousingReader_AS17_Latch_and_Error_Clear_Control_Bits_1;
	HwOutputs.HousingReader_AS17_Operation_instruction_Control_Bits_1 := PlcOutputs.HousingReader_AS17_Operation_instruction_Control_Bits_1;
	HwOutputs.HousingReader_AS17_Completion_Clear_Control_Bits_1 := PlcOutputs.HousingReader_AS17_Completion_Clear_Control_Bits_1;
	HwOutputs.HousingReader_AS17_Parameter_Bank_Number_1 := PlcOutputs.HousingReader_AS17_Parameter_Bank_Number_1;
	HwOutputs.HousingReader_AS17_User_Data_128Byte_1[0] := PlcOutputs.HousingReader_AS17_User_Data_128Byte_1[0];
	HwOutputs.HousingReader_AS17_User_Data_128Byte_1[1] := PlcOutputs.HousingReader_AS17_User_Data_128Byte_1[1];
	HwOutputs.HousingReader_AS17_User_Data_128Byte_1[2] := PlcOutputs.HousingReader_AS17_User_Data_128Byte_1[2];
	HwOutputs.HousingReader_AS17_User_Data_128Byte_1[3] := PlcOutputs.HousingReader_AS17_User_Data_128Byte_1[3];
	HwOutputs.HousingReader_AS17_User_Data_128Byte_1[4] := PlcOutputs.HousingReader_AS17_User_Data_128Byte_1[4];
	HwOutputs.HousingReader_AS17_User_Data_128Byte_1[5] := PlcOutputs.HousingReader_AS17_User_Data_128Byte_1[5];
	HwOutputs.HousingReader_AS17_User_Data_128Byte_1[6] := PlcOutputs.HousingReader_AS17_User_Data_128Byte_1[6];
	HwOutputs.HousingReader_AS17_User_Data_128Byte_1[7] := PlcOutputs.HousingReader_AS17_User_Data_128Byte_1[7];
	HwOutputs.HousingReader_AS17_User_Data_128Byte_1[8] := PlcOutputs.HousingReader_AS17_User_Data_128Byte_1[8];
	HwOutputs.HousingReader_AS17_User_Data_128Byte_1[9] := PlcOutputs.HousingReader_AS17_User_Data_128Byte_1[9];
	HwOutputs.HousingReader_AS17_User_Data_128Byte_1[10] := PlcOutputs.HousingReader_AS17_User_Data_128Byte_1[10];
	HwOutputs.HousingReader_AS17_User_Data_128Byte_1[11] := PlcOutputs.HousingReader_AS17_User_Data_128Byte_1[11];
	HwOutputs.HousingReader_AS17_User_Data_128Byte_1[12] := PlcOutputs.HousingReader_AS17_User_Data_128Byte_1[12];
	HwOutputs.HousingReader_AS17_User_Data_128Byte_1[13] := PlcOutputs.HousingReader_AS17_User_Data_128Byte_1[13];
	HwOutputs.HousingReader_AS17_User_Data_128Byte_1[14] := PlcOutputs.HousingReader_AS17_User_Data_128Byte_1[14];
	HwOutputs.HousingReader_AS17_User_Data_128Byte_1[15] := PlcOutputs.HousingReader_AS17_User_Data_128Byte_1[15];
	HwOutputs.HousingReader_AS17_User_Data_128Byte_1[16] := PlcOutputs.HousingReader_AS17_User_Data_128Byte_1[16];
	HwOutputs.HousingReader_AS17_User_Data_128Byte_1[17] := PlcOutputs.HousingReader_AS17_User_Data_128Byte_1[17];
	HwOutputs.HousingReader_AS17_User_Data_128Byte_1[18] := PlcOutputs.HousingReader_AS17_User_Data_128Byte_1[18];
	HwOutputs.HousingReader_AS17_User_Data_128Byte_1[19] := PlcOutputs.HousingReader_AS17_User_Data_128Byte_1[19];
	HwOutputs.HousingReader_AS17_User_Data_128Byte_1[20] := PlcOutputs.HousingReader_AS17_User_Data_128Byte_1[20];
	HwOutputs.HousingReader_AS17_User_Data_128Byte_1[21] := PlcOutputs.HousingReader_AS17_User_Data_128Byte_1[21];
	HwOutputs.HousingReader_AS17_User_Data_128Byte_1[22] := PlcOutputs.HousingReader_AS17_User_Data_128Byte_1[22];
	HwOutputs.HousingReader_AS17_User_Data_128Byte_1[23] := PlcOutputs.HousingReader_AS17_User_Data_128Byte_1[23];
	HwOutputs.HousingReader_AS17_User_Data_128Byte_1[24] := PlcOutputs.HousingReader_AS17_User_Data_128Byte_1[24];
	HwOutputs.HousingReader_AS17_User_Data_128Byte_1[25] := PlcOutputs.HousingReader_AS17_User_Data_128Byte_1[25];
	HwOutputs.HousingReader_AS17_User_Data_128Byte_1[26] := PlcOutputs.HousingReader_AS17_User_Data_128Byte_1[26];
	HwOutputs.HousingReader_AS17_User_Data_128Byte_1[27] := PlcOutputs.HousingReader_AS17_User_Data_128Byte_1[27];
	HwOutputs.HousingReader_AS17_User_Data_128Byte_1[28] := PlcOutputs.HousingReader_AS17_User_Data_128Byte_1[28];
	HwOutputs.HousingReader_AS17_User_Data_128Byte_1[29] := PlcOutputs.HousingReader_AS17_User_Data_128Byte_1[29];
	HwOutputs.HousingReader_AS17_User_Data_128Byte_1[30] := PlcOutputs.HousingReader_AS17_User_Data_128Byte_1[30];
	HwOutputs.HousingReader_AS17_User_Data_128Byte_1[31] := PlcOutputs.HousingReader_AS17_User_Data_128Byte_1[31];
	HwOutputs.HousingReader_AS17_User_Data_128Byte_1[32] := PlcOutputs.HousingReader_AS17_User_Data_128Byte_1[32];
	HwOutputs.HousingReader_AS17_User_Data_128Byte_1[33] := PlcOutputs.HousingReader_AS17_User_Data_128Byte_1[33];
	HwOutputs.HousingReader_AS17_User_Data_128Byte_1[34] := PlcOutputs.HousingReader_AS17_User_Data_128Byte_1[34];
	HwOutputs.HousingReader_AS17_User_Data_128Byte_1[35] := PlcOutputs.HousingReader_AS17_User_Data_128Byte_1[35];
	HwOutputs.HousingReader_AS17_User_Data_128Byte_1[36] := PlcOutputs.HousingReader_AS17_User_Data_128Byte_1[36];
	HwOutputs.HousingReader_AS17_User_Data_128Byte_1[37] := PlcOutputs.HousingReader_AS17_User_Data_128Byte_1[37];
	HwOutputs.HousingReader_AS17_User_Data_128Byte_1[38] := PlcOutputs.HousingReader_AS17_User_Data_128Byte_1[38];
	HwOutputs.HousingReader_AS17_User_Data_128Byte_1[39] := PlcOutputs.HousingReader_AS17_User_Data_128Byte_1[39];
	HwOutputs.HousingReader_AS17_User_Data_128Byte_1[40] := PlcOutputs.HousingReader_AS17_User_Data_128Byte_1[40];
	HwOutputs.HousingReader_AS17_User_Data_128Byte_1[41] := PlcOutputs.HousingReader_AS17_User_Data_128Byte_1[41];
	HwOutputs.HousingReader_AS17_User_Data_128Byte_1[42] := PlcOutputs.HousingReader_AS17_User_Data_128Byte_1[42];
	HwOutputs.HousingReader_AS17_User_Data_128Byte_1[43] := PlcOutputs.HousingReader_AS17_User_Data_128Byte_1[43];
	HwOutputs.HousingReader_AS17_User_Data_128Byte_1[44] := PlcOutputs.HousingReader_AS17_User_Data_128Byte_1[44];
	HwOutputs.HousingReader_AS17_User_Data_128Byte_1[45] := PlcOutputs.HousingReader_AS17_User_Data_128Byte_1[45];
	HwOutputs.HousingReader_AS17_User_Data_128Byte_1[46] := PlcOutputs.HousingReader_AS17_User_Data_128Byte_1[46];
	HwOutputs.HousingReader_AS17_User_Data_128Byte_1[47] := PlcOutputs.HousingReader_AS17_User_Data_128Byte_1[47];
	HwOutputs.HousingReader_AS17_User_Data_128Byte_1[48] := PlcOutputs.HousingReader_AS17_User_Data_128Byte_1[48];
	HwOutputs.HousingReader_AS17_User_Data_128Byte_1[49] := PlcOutputs.HousingReader_AS17_User_Data_128Byte_1[49];
	HwOutputs.HousingReader_AS17_User_Data_128Byte_1[50] := PlcOutputs.HousingReader_AS17_User_Data_128Byte_1[50];
	HwOutputs.HousingReader_AS17_User_Data_128Byte_1[51] := PlcOutputs.HousingReader_AS17_User_Data_128Byte_1[51];
	HwOutputs.HousingReader_AS17_User_Data_128Byte_1[52] := PlcOutputs.HousingReader_AS17_User_Data_128Byte_1[52];
	HwOutputs.HousingReader_AS17_User_Data_128Byte_1[53] := PlcOutputs.HousingReader_AS17_User_Data_128Byte_1[53];
	HwOutputs.HousingReader_AS17_User_Data_128Byte_1[54] := PlcOutputs.HousingReader_AS17_User_Data_128Byte_1[54];
	HwOutputs.HousingReader_AS17_User_Data_128Byte_1[55] := PlcOutputs.HousingReader_AS17_User_Data_128Byte_1[55];
	HwOutputs.HousingReader_AS17_User_Data_128Byte_1[56] := PlcOutputs.HousingReader_AS17_User_Data_128Byte_1[56];
	HwOutputs.HousingReader_AS17_User_Data_128Byte_1[57] := PlcOutputs.HousingReader_AS17_User_Data_128Byte_1[57];
	HwOutputs.HousingReader_AS17_User_Data_128Byte_1[58] := PlcOutputs.HousingReader_AS17_User_Data_128Byte_1[58];
	HwOutputs.HousingReader_AS17_User_Data_128Byte_1[59] := PlcOutputs.HousingReader_AS17_User_Data_128Byte_1[59];
	HwOutputs.HousingReader_AS17_User_Data_128Byte_1[60] := PlcOutputs.HousingReader_AS17_User_Data_128Byte_1[60];
	HwOutputs.HousingReader_AS17_User_Data_128Byte_1[61] := PlcOutputs.HousingReader_AS17_User_Data_128Byte_1[61];
	HwOutputs.HousingReader_AS17_User_Data_128Byte_1[62] := PlcOutputs.HousingReader_AS17_User_Data_128Byte_1[62];
	HwOutputs.HousingReader_AS17_User_Data_128Byte_1[63] := PlcOutputs.HousingReader_AS17_User_Data_128Byte_1[63];
	HwOutputs.HousingReader_AS17_User_Data_128Byte_1[64] := PlcOutputs.HousingReader_AS17_User_Data_128Byte_1[64];
	HwOutputs.HousingReader_AS17_User_Data_128Byte_1[65] := PlcOutputs.HousingReader_AS17_User_Data_128Byte_1[65];
	HwOutputs.HousingReader_AS17_User_Data_128Byte_1[66] := PlcOutputs.HousingReader_AS17_User_Data_128Byte_1[66];
	HwOutputs.HousingReader_AS17_User_Data_128Byte_1[67] := PlcOutputs.HousingReader_AS17_User_Data_128Byte_1[67];
	HwOutputs.HousingReader_AS17_User_Data_128Byte_1[68] := PlcOutputs.HousingReader_AS17_User_Data_128Byte_1[68];
	HwOutputs.HousingReader_AS17_User_Data_128Byte_1[69] := PlcOutputs.HousingReader_AS17_User_Data_128Byte_1[69];
	HwOutputs.HousingReader_AS17_User_Data_128Byte_1[70] := PlcOutputs.HousingReader_AS17_User_Data_128Byte_1[70];
	HwOutputs.HousingReader_AS17_User_Data_128Byte_1[71] := PlcOutputs.HousingReader_AS17_User_Data_128Byte_1[71];
	HwOutputs.HousingReader_AS17_User_Data_128Byte_1[72] := PlcOutputs.HousingReader_AS17_User_Data_128Byte_1[72];
	HwOutputs.HousingReader_AS17_User_Data_128Byte_1[73] := PlcOutputs.HousingReader_AS17_User_Data_128Byte_1[73];
	HwOutputs.HousingReader_AS17_User_Data_128Byte_1[74] := PlcOutputs.HousingReader_AS17_User_Data_128Byte_1[74];
	HwOutputs.HousingReader_AS17_User_Data_128Byte_1[75] := PlcOutputs.HousingReader_AS17_User_Data_128Byte_1[75];
	HwOutputs.HousingReader_AS17_User_Data_128Byte_1[76] := PlcOutputs.HousingReader_AS17_User_Data_128Byte_1[76];
	HwOutputs.HousingReader_AS17_User_Data_128Byte_1[77] := PlcOutputs.HousingReader_AS17_User_Data_128Byte_1[77];
	HwOutputs.HousingReader_AS17_User_Data_128Byte_1[78] := PlcOutputs.HousingReader_AS17_User_Data_128Byte_1[78];
	HwOutputs.HousingReader_AS17_User_Data_128Byte_1[79] := PlcOutputs.HousingReader_AS17_User_Data_128Byte_1[79];
	HwOutputs.HousingReader_AS17_User_Data_128Byte_1[80] := PlcOutputs.HousingReader_AS17_User_Data_128Byte_1[80];
	HwOutputs.HousingReader_AS17_User_Data_128Byte_1[81] := PlcOutputs.HousingReader_AS17_User_Data_128Byte_1[81];
	HwOutputs.HousingReader_AS17_User_Data_128Byte_1[82] := PlcOutputs.HousingReader_AS17_User_Data_128Byte_1[82];
	HwOutputs.HousingReader_AS17_User_Data_128Byte_1[83] := PlcOutputs.HousingReader_AS17_User_Data_128Byte_1[83];
	HwOutputs.HousingReader_AS17_User_Data_128Byte_1[84] := PlcOutputs.HousingReader_AS17_User_Data_128Byte_1[84];
	HwOutputs.HousingReader_AS17_User_Data_128Byte_1[85] := PlcOutputs.HousingReader_AS17_User_Data_128Byte_1[85];
	HwOutputs.HousingReader_AS17_User_Data_128Byte_1[86] := PlcOutputs.HousingReader_AS17_User_Data_128Byte_1[86];
	HwOutputs.HousingReader_AS17_User_Data_128Byte_1[87] := PlcOutputs.HousingReader_AS17_User_Data_128Byte_1[87];
	HwOutputs.HousingReader_AS17_User_Data_128Byte_1[88] := PlcOutputs.HousingReader_AS17_User_Data_128Byte_1[88];
	HwOutputs.HousingReader_AS17_User_Data_128Byte_1[89] := PlcOutputs.HousingReader_AS17_User_Data_128Byte_1[89];
	HwOutputs.HousingReader_AS17_User_Data_128Byte_1[90] := PlcOutputs.HousingReader_AS17_User_Data_128Byte_1[90];
	HwOutputs.HousingReader_AS17_User_Data_128Byte_1[91] := PlcOutputs.HousingReader_AS17_User_Data_128Byte_1[91];
	HwOutputs.HousingReader_AS17_User_Data_128Byte_1[92] := PlcOutputs.HousingReader_AS17_User_Data_128Byte_1[92];
	HwOutputs.HousingReader_AS17_User_Data_128Byte_1[93] := PlcOutputs.HousingReader_AS17_User_Data_128Byte_1[93];
	HwOutputs.HousingReader_AS17_User_Data_128Byte_1[94] := PlcOutputs.HousingReader_AS17_User_Data_128Byte_1[94];
	HwOutputs.HousingReader_AS17_User_Data_128Byte_1[95] := PlcOutputs.HousingReader_AS17_User_Data_128Byte_1[95];
	HwOutputs.HousingReader_AS17_User_Data_128Byte_1[96] := PlcOutputs.HousingReader_AS17_User_Data_128Byte_1[96];
	HwOutputs.HousingReader_AS17_User_Data_128Byte_1[97] := PlcOutputs.HousingReader_AS17_User_Data_128Byte_1[97];
	HwOutputs.HousingReader_AS17_User_Data_128Byte_1[98] := PlcOutputs.HousingReader_AS17_User_Data_128Byte_1[98];
	HwOutputs.HousingReader_AS17_User_Data_128Byte_1[99] := PlcOutputs.HousingReader_AS17_User_Data_128Byte_1[99];
	HwOutputs.HousingReader_AS17_User_Data_128Byte_1[100] := PlcOutputs.HousingReader_AS17_User_Data_128Byte_1[100];
	HwOutputs.HousingReader_AS17_User_Data_128Byte_1[101] := PlcOutputs.HousingReader_AS17_User_Data_128Byte_1[101];
	HwOutputs.HousingReader_AS17_User_Data_128Byte_1[102] := PlcOutputs.HousingReader_AS17_User_Data_128Byte_1[102];
	HwOutputs.HousingReader_AS17_User_Data_128Byte_1[103] := PlcOutputs.HousingReader_AS17_User_Data_128Byte_1[103];
	HwOutputs.HousingReader_AS17_User_Data_128Byte_1[104] := PlcOutputs.HousingReader_AS17_User_Data_128Byte_1[104];
	HwOutputs.HousingReader_AS17_User_Data_128Byte_1[105] := PlcOutputs.HousingReader_AS17_User_Data_128Byte_1[105];
	HwOutputs.HousingReader_AS17_User_Data_128Byte_1[106] := PlcOutputs.HousingReader_AS17_User_Data_128Byte_1[106];
	HwOutputs.HousingReader_AS17_User_Data_128Byte_1[107] := PlcOutputs.HousingReader_AS17_User_Data_128Byte_1[107];
	HwOutputs.HousingReader_AS17_User_Data_128Byte_1[108] := PlcOutputs.HousingReader_AS17_User_Data_128Byte_1[108];
	HwOutputs.HousingReader_AS17_User_Data_128Byte_1[109] := PlcOutputs.HousingReader_AS17_User_Data_128Byte_1[109];
	HwOutputs.HousingReader_AS17_User_Data_128Byte_1[110] := PlcOutputs.HousingReader_AS17_User_Data_128Byte_1[110];
	HwOutputs.HousingReader_AS17_User_Data_128Byte_1[111] := PlcOutputs.HousingReader_AS17_User_Data_128Byte_1[111];
	HwOutputs.HousingReader_AS17_User_Data_128Byte_1[112] := PlcOutputs.HousingReader_AS17_User_Data_128Byte_1[112];
	HwOutputs.HousingReader_AS17_User_Data_128Byte_1[113] := PlcOutputs.HousingReader_AS17_User_Data_128Byte_1[113];
	HwOutputs.HousingReader_AS17_User_Data_128Byte_1[114] := PlcOutputs.HousingReader_AS17_User_Data_128Byte_1[114];
	HwOutputs.HousingReader_AS17_User_Data_128Byte_1[115] := PlcOutputs.HousingReader_AS17_User_Data_128Byte_1[115];
	HwOutputs.HousingReader_AS17_User_Data_128Byte_1[116] := PlcOutputs.HousingReader_AS17_User_Data_128Byte_1[116];
	HwOutputs.HousingReader_AS17_User_Data_128Byte_1[117] := PlcOutputs.HousingReader_AS17_User_Data_128Byte_1[117];
	HwOutputs.HousingReader_AS17_User_Data_128Byte_1[118] := PlcOutputs.HousingReader_AS17_User_Data_128Byte_1[118];
	HwOutputs.HousingReader_AS17_User_Data_128Byte_1[119] := PlcOutputs.HousingReader_AS17_User_Data_128Byte_1[119];
	HwOutputs.HousingReader_AS17_User_Data_128Byte_1[120] := PlcOutputs.HousingReader_AS17_User_Data_128Byte_1[120];
	HwOutputs.HousingReader_AS17_User_Data_128Byte_1[121] := PlcOutputs.HousingReader_AS17_User_Data_128Byte_1[121];
	HwOutputs.HousingReader_AS17_User_Data_128Byte_1[122] := PlcOutputs.HousingReader_AS17_User_Data_128Byte_1[122];
	HwOutputs.HousingReader_AS17_User_Data_128Byte_1[123] := PlcOutputs.HousingReader_AS17_User_Data_128Byte_1[123];
	HwOutputs.HousingReader_AS17_User_Data_128Byte_1[124] := PlcOutputs.HousingReader_AS17_User_Data_128Byte_1[124];
	HwOutputs.HousingReader_AS17_User_Data_128Byte_1[125] := PlcOutputs.HousingReader_AS17_User_Data_128Byte_1[125];
	HwOutputs.HousingReader_AS17_User_Data_128Byte_1[126] := PlcOutputs.HousingReader_AS17_User_Data_128Byte_1[126];
	HwOutputs.HousingReader_AS17_User_Data_128Byte_1[127] := PlcOutputs.HousingReader_AS17_User_Data_128Byte_1[127];
	HwOutputs.HousingReader_AS17_User_Data_128Byte_1[128] := PlcOutputs.HousingReader_AS17_User_Data_128Byte_1[128];
	HwOutputs.HousingReader_AS17_User_Data_128Byte_1[129] := PlcOutputs.HousingReader_AS17_User_Data_128Byte_1[129];
	HwOutputs.CPX_PneuOst_AS17_MPA1S_VMPA1_FB_EMS_8_8DO_1 := PlcOutputs.CPX_PneuOst_AS17_MPA1S_VMPA1_FB_EMS_8_8DO_1;
	HwOutputs.CPX_PneuOst_AS17_MPA1S_VMPA1_FB_EMS_8_8DO_2 := PlcOutputs.CPX_PneuOst_AS17_MPA1S_VMPA1_FB_EMS_8_8DO_2;
	HwOutputs.CPX_PneuOst_AS17_MPA1S_VMPA1_FB_EMS_8_8DO_3 := PlcOutputs.CPX_PneuOst_AS17_MPA1S_VMPA1_FB_EMS_8_8DO_3;
	HwOutputs.CPX_PneuOst_AS17_MPA1S_VMPA1_FB_EMS_8_8DO_4 := PlcOutputs.CPX_PneuOst_AS17_MPA1S_VMPA1_FB_EMS_8_8DO_4;
	HwOutputs.CPX_PneuOst_AS17_MPA1G_VMPA1_FB_EMG_8_8DO_1 := PlcOutputs.CPX_PneuOst_AS17_MPA1G_VMPA1_FB_EMG_8_8DO_1;
	HwOutputs.SEW_AS_1_Drive_1x3PD_1[0] := PlcOutputs.SEW_AS_1_Drive_1x3PD_1[0];
	HwOutputs.SEW_AS_1_Drive_1x3PD_1[1] := PlcOutputs.SEW_AS_1_Drive_1x3PD_1[1];
	HwOutputs.SEW_AS_1_Drive_1x3PD_1[2] := PlcOutputs.SEW_AS_1_Drive_1x3PD_1[2];
	HwOutputs.SEW_AS_1_Drive_1x3PD_1[3] := PlcOutputs.SEW_AS_1_Drive_1x3PD_1[3];
	HwOutputs.SEW_AS_1_Drive_1x3PD_1[4] := PlcOutputs.SEW_AS_1_Drive_1x3PD_1[4];
	HwOutputs.SEW_AS_1_Drive_1x3PD_1[5] := PlcOutputs.SEW_AS_1_Drive_1x3PD_1[5];
	HwOutputs.Glue_DO_16_bytes_1[0] := PlcOutputs.Glue_DO_16_bytes_1[0];
	HwOutputs.Glue_DO_16_bytes_1[1] := PlcOutputs.Glue_DO_16_bytes_1[1];
	HwOutputs.Glue_DO_16_bytes_1[2] := PlcOutputs.Glue_DO_16_bytes_1[2];
	HwOutputs.Glue_DO_16_bytes_1[3] := PlcOutputs.Glue_DO_16_bytes_1[3];
	HwOutputs.Glue_DO_16_bytes_1[4] := PlcOutputs.Glue_DO_16_bytes_1[4];
	HwOutputs.Glue_DO_16_bytes_1[5] := PlcOutputs.Glue_DO_16_bytes_1[5];
	HwOutputs.Glue_DO_16_bytes_1[6] := PlcOutputs.Glue_DO_16_bytes_1[6];
	HwOutputs.Glue_DO_16_bytes_1[7] := PlcOutputs.Glue_DO_16_bytes_1[7];
	HwOutputs.Glue_DO_16_bytes_1[8] := PlcOutputs.Glue_DO_16_bytes_1[8];
	HwOutputs.Glue_DO_16_bytes_1[9] := PlcOutputs.Glue_DO_16_bytes_1[9];
	HwOutputs.Glue_DO_16_bytes_1[10] := PlcOutputs.Glue_DO_16_bytes_1[10];
	HwOutputs.Glue_DO_16_bytes_1[11] := PlcOutputs.Glue_DO_16_bytes_1[11];
	HwOutputs.Glue_DO_16_bytes_1[12] := PlcOutputs.Glue_DO_16_bytes_1[12];
	HwOutputs.Glue_DO_16_bytes_1[13] := PlcOutputs.Glue_DO_16_bytes_1[13];
	HwOutputs.Glue_DO_16_bytes_1[14] := PlcOutputs.Glue_DO_16_bytes_1[14];
	HwOutputs.Glue_DO_16_bytes_1[15] := PlcOutputs.Glue_DO_16_bytes_1[15];
END_FUNCTION
